PROGRAM idle
VAR
	ed_routine_idle: BOOL;
	redox_doser_idle_enable: BOOL;
	
	tmr_idle_pumps: TON;
	u_3112_idle_request: BOOL;
	u_3312_idle_request: BOOL;
	u_3405_idle_request: BOOL;
	u_3212_idle_request: BOOL;
	tmr_idle_pump_delay: TON;
	u_3112_running: BOOL;
	u_3112_speed_ref: INT;
	u_3112_sp: REAL;
	salt_pressure_actual: REAL;
	u_3112_ready: BOOL;
	u_3212_running: BOOL;
	u_3212_ready: BOOL;
	u_3312_ready: BOOL;
	u_3312_running: BOOL;
	u_3405_running: BOOL;
	u_3405_ready: BOOL;
	stack_power_enable: BOOL;
	nv_3110_open_request: BOOL;
	nv_3210_open_request: BOOL;
	nv_3310_open_request: BOOL;
	nv_3110_open_feedback: BOOL;
	nv_3210_open_feedback: BOOL;
	nv_3310_open_feedback: BOOL;
	nv_3110_idle_request: BOOL;
	nv_3210_idle_request: BOOL;
	nv_3310_idle_request: BOOL;
	nv_3135_idle_request: BOOL;
	nv_3235_idle_request: BOOL;
	nv_3335_idle_request: BOOL;
	nv_3372_idle_request: BOOL;
	nv_3162_idle_request: BOOL;

	idle_stack_power_enable: BOOL;
	idle_TEMP_BIT: BOOL;
	tmr_idle_valye_delay: TON;
	tmr_idle_valve_delay: TON;
	tmr_idle_valve_delay_et: TIME;
	tmr_idle_valve_delay_q: BOOL;
	u_3112_idle_pressure_setpoint_request: REAL;
	u_3212_idle_pressure_setpoint_request: REAL;
	u_3312_idle_pressure_setpoint_request: REAL;
	u_3405_idle_pressure_setpoint_request: REAL;
END_VAR
VAR // added by the converter: edge detectors and wires of the graphical bodies
    _w1, _w2 : BOOL;
END_VAR

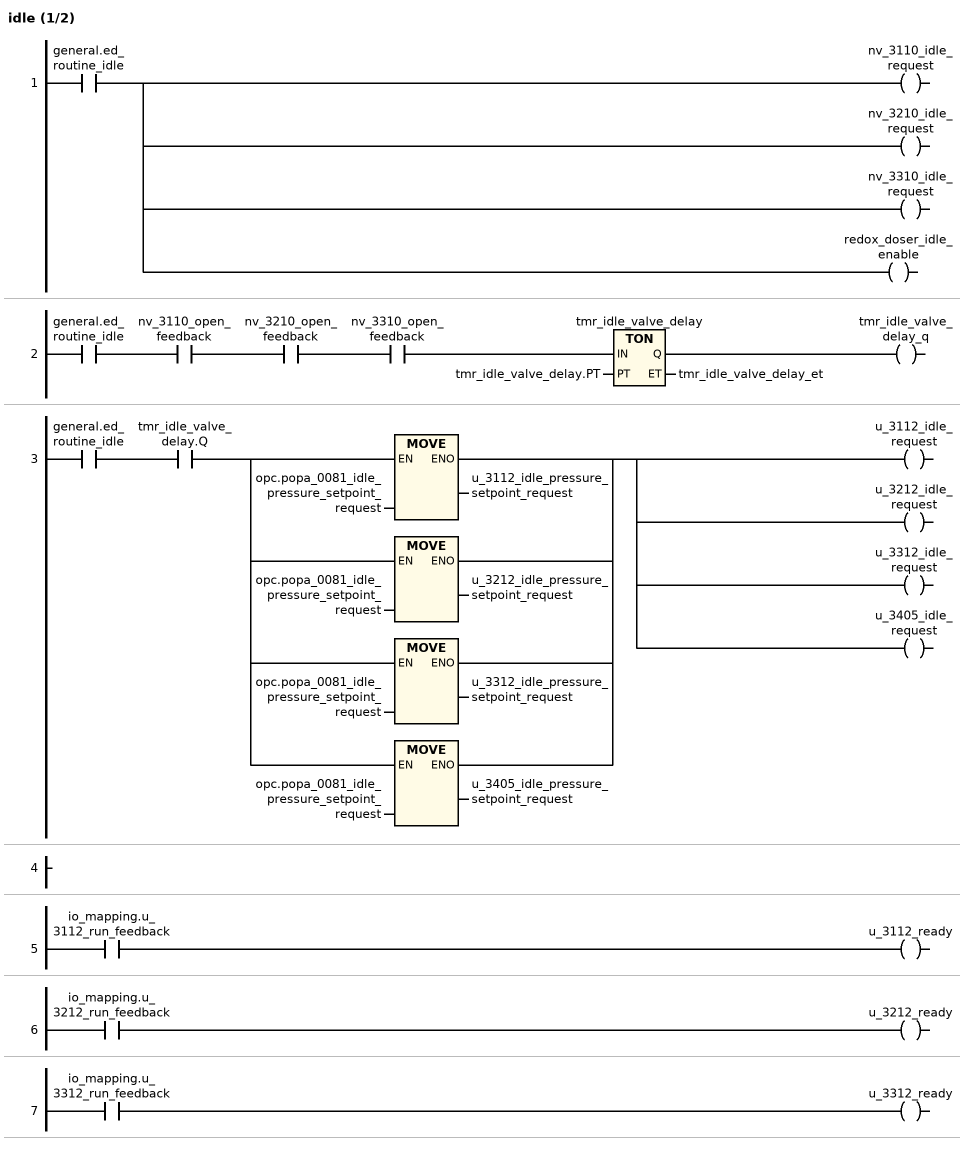
// NETWORK 1
nv_3110_idle_request := general.ed_routine_idle;
nv_3210_idle_request := general.ed_routine_idle;
nv_3310_idle_request := general.ed_routine_idle;
redox_doser_idle_enable := general.ed_routine_idle;

// NETWORK 2
tmr_idle_valve_delay(
    IN := general.ed_routine_idle AND nv_3110_open_feedback AND nv_3210_open_feedback AND nv_3310_open_feedback,
    PT := tmr_idle_valve_delay.PT,
    ET => tmr_idle_valve_delay_et); // TON
tmr_idle_valve_delay_q := tmr_idle_valve_delay.Q;

// NETWORK 3
_w1 := general.ed_routine_idle AND tmr_idle_valve_delay.Q;
IF _w1 THEN u_3112_idle_pressure_setpoint_request := opc.popa_0081_idle_pressure_setpoint_request; END_IF
IF _w1 THEN u_3212_idle_pressure_setpoint_request := opc.popa_0081_idle_pressure_setpoint_request; END_IF
IF _w1 THEN u_3312_idle_pressure_setpoint_request := opc.popa_0081_idle_pressure_setpoint_request; END_IF
IF _w1 THEN u_3405_idle_pressure_setpoint_request := opc.popa_0081_idle_pressure_setpoint_request; END_IF
_w2 := _w1 OR (_w1 OR (_w1 OR _w1));
u_3112_idle_request := _w2;
u_3212_idle_request := _w2;
u_3312_idle_request := _w2;
u_3405_idle_request := _w2;

// NETWORK 4

// NETWORK 5
u_3112_ready := io_mapping.u_3112_run_feedback;

// NETWORK 6
u_3212_ready := io_mapping.u_3212_run_feedback;

// NETWORK 7
u_3312_ready := io_mapping.u_3312_run_feedback;

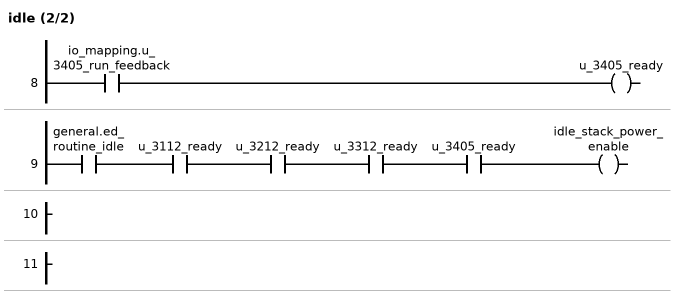
// NETWORK 8
u_3405_ready := io_mapping.u_3405_run_feedback;

// NETWORK 9
idle_stack_power_enable := general.ed_routine_idle AND u_3112_ready AND u_3212_ready AND u_3312_ready AND u_3405_ready;

// NETWORK 10

// NETWORK 11

END_PROGRAM

(* stored: Version 1.1.0.1, ProductVersion 3.1.4024.12
   POU idle: Id {3d08b1fd-a23f-437d-8121-cefd84a9c392}, SpecialFunc None *)
